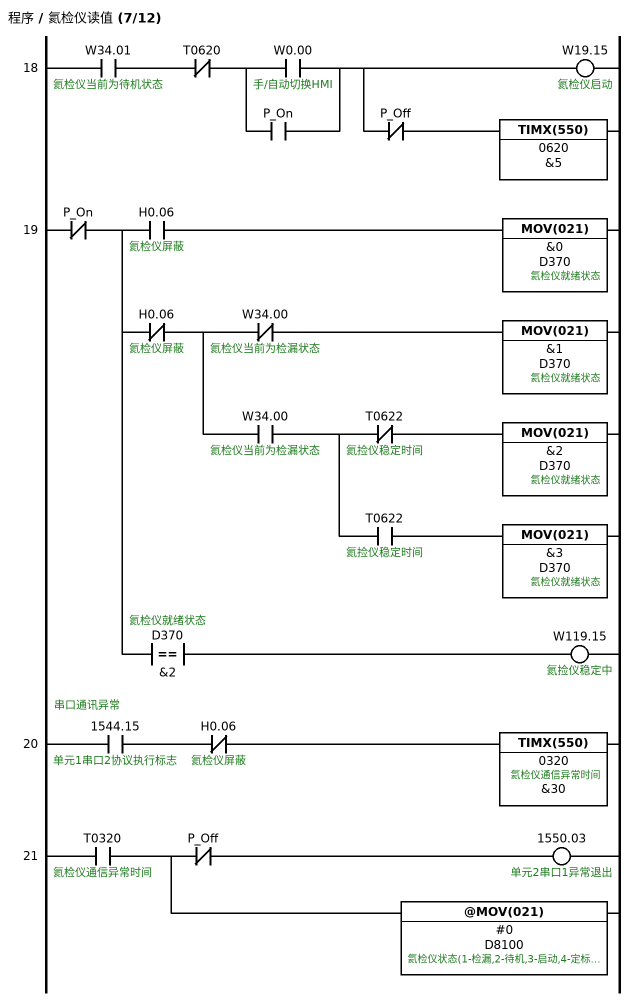
; [picture p168: 程序 / 氦检仪读值, rungs 18-21]
; rung 18
LD W34.01  ; 氦检仪当前为待机状态
ANDNOT T0620
LD W0.00  ; 手/自动切换HMI
OR P_On
ANDLD
OUT W19.15  ; 氦检仪启动
ANDNOT P_Off
TIMX(550) 0620 &5
; rung 19
LDNOT P_On
OUT TR0
AND H0.06  ; 氦检仪屏蔽
MOV(021) &0 D370  ; 氦检仪就绪状态
LD TR0
ANDNOT H0.06  ; 氦检仪屏蔽
OUT TR1
ANDNOT W34.00  ; 氦检仪当前为检漏状态
MOV(021) &1 D370  ; 氦检仪就绪状态
LD TR1
AND W34.00  ; 氦检仪当前为检漏状态
OUT TR1
ANDNOT T0622  ; 氦捡仪稳定时间
MOV(021) &2 D370  ; 氦检仪就绪状态
LD TR1
AND T0622  ; 氦捡仪稳定时间
MOV(021) &3 D370  ; 氦检仪就绪状态
LD TR0
AND=(300) D370 &2  ; 氦检仪就绪状态
OUT W119.15  ; 氦捡仪稳定中
; rung 20: 串口通讯异常
LD 1544.15  ; 单元1串口2协议执行标志
ANDNOT H0.06  ; 氦检仪屏蔽
TIMX(550) 0320 &30  ; 氦检仪通信异常时间
; rung 21
LD T0320  ; 氦检仪通信异常时间
OUT TR0
ANDNOT P_Off
OUT 1550.03  ; 单元2串口1异常退出
LD TR0
@MOV(021) #0 D8100  ; 氦检仪状态(1-检漏,2-待机,3-启动,4-定标,5-错误,6-暂停)

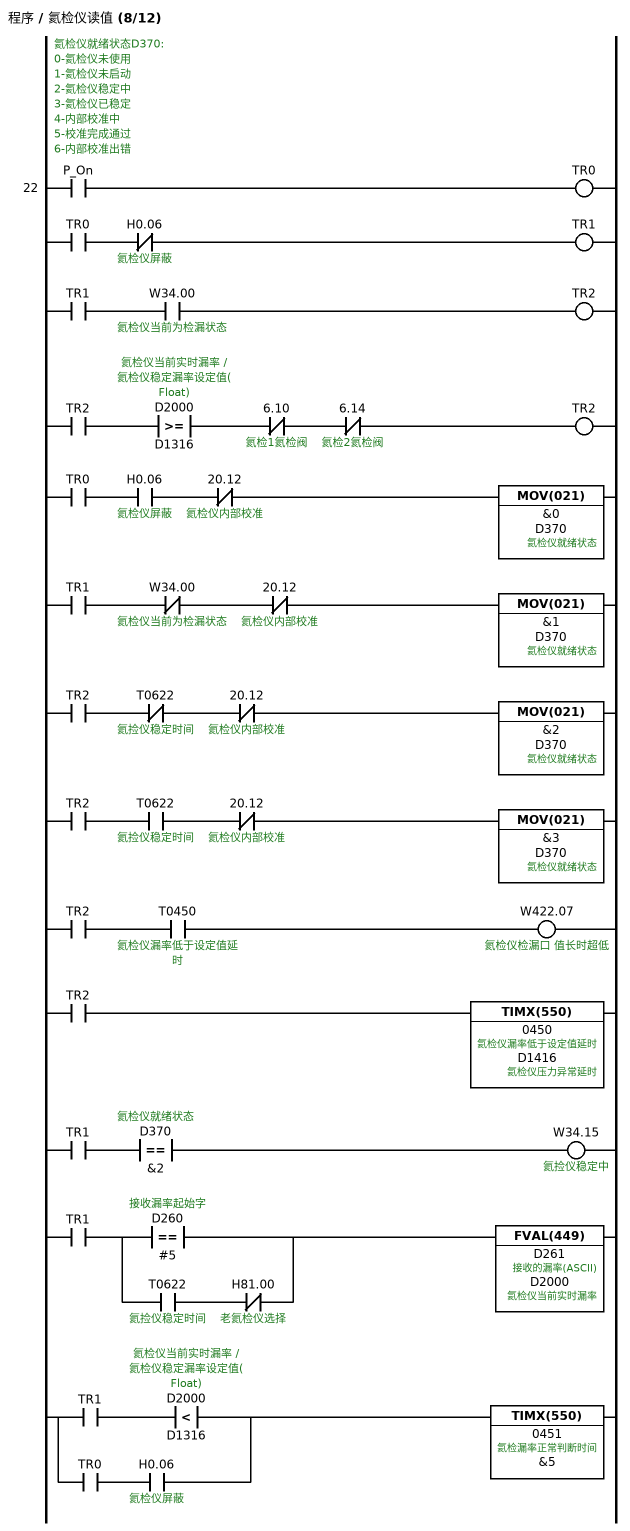
; rung 22: 氦检仪就绪状态D370: / 0-氦检仪未使用 / 1-氦检仪未启动 / 2-氦检仪稳定中 / 3-氦检仪已稳定 / 4-内部校准中 / 5-校准完成通过 / 6-内部校准出错
LD P_On
OUT TR0
AND H0.06  ; 氦检仪屏蔽
ANDNOT 20.12  ; 氦检仪内部校准
MOV(021) &0 D370  ; 氦检仪就绪状态
LD TR0
ANDNOT H0.06  ; 氦检仪屏蔽
OUT TR1
ANDNOT W34.00  ; 氦检仪当前为检漏状态
ANDNOT 20.12  ; 氦检仪内部校准
MOV(021) &1 D370  ; 氦检仪就绪状态
LD TR1
AND W34.00  ; 氦检仪当前为检漏状态
OUT TR2
ANDNOT T0622  ; 氦捡仪稳定时间
ANDNOT 20.12  ; 氦检仪内部校准
MOV(021) &2 D370  ; 氦检仪就绪状态
LD TR2
AND T0622  ; 氦捡仪稳定时间
ANDNOT 20.12  ; 氦检仪内部校准
MOV(021) &3 D370  ; 氦检仪就绪状态
LD TR2
AND>=F(334) D2000 D1316  ; 氦检仪当前实时漏率, 氦检仪稳定漏率设定值(Float)
ANDNOT 6.10  ; 氦检1氦检阀
ANDNOT 6.14  ; 氦检2氦检阀
OUT TR2
AND T0450  ; 氦检仪漏率低于设定值延时
OUT W422.07  ; 氦检仪检漏口 值长时超低
LD TR2
TIMX(550) 0450 D1416  ; 氦检仪压力异常延时, 氦检仪漏率低于设定值延时
LD TR1
AND=(300) D370 &2  ; 氦检仪就绪状态
OUT W34.15  ; 氦捡仪稳定中
LD TR1
LD=(300) D260 #5  ; 接收漏率起始字
LD T0622  ; 氦捡仪稳定时间
ANDNOT H81.00  ; 老氦检仪选择
ORLD
ANDLD
FVAL(449) D261 D2000  ; 接收的漏率(ASCII), 氦检仪当前实时漏率
LD TR1
AND<F(331) D2000 D1316  ; 氦检仪当前实时漏率, 氦检仪稳定漏率设定值(Float)
LD TR0
AND H0.06  ; 氦检仪屏蔽
ORLD
TIMX(550) 0451 &5  ; 氦检漏率正常判断时间

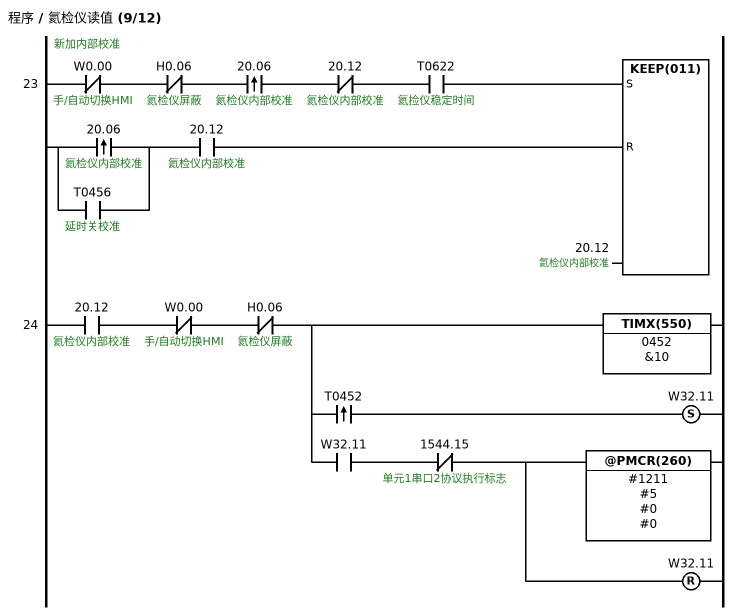
; rung 23: 新加内部校准
LDNOT W0.00  ; 手/自动切换HMI
ANDNOT H0.06  ; 氦检仪屏蔽
@AND 20.06  ; 氦检仪内部校准
ANDNOT 20.12  ; 氦检仪内部校准
AND T0622  ; 氦捡仪稳定时间
@LD 20.06  ; 氦检仪内部校准
OR T0456  ; 延时关校准
AND 20.12  ; 氦检仪内部校准
KEEP(011) 20.12  ; 氦检仪内部校准
; rung 24
LD 20.12  ; 氦检仪内部校准
ANDNOT W0.00  ; 手/自动切换HMI
ANDNOT H0.06  ; 氦检仪屏蔽
OUT TR0
TIMX(550) 0452 &10
@AND T0452
SET W32.11
LD TR0
AND W32.11
ANDNOT 1544.15  ; 单元1串口2协议执行标志
@PMCR(260) #1211 #5 #0 #0
RSET W32.11

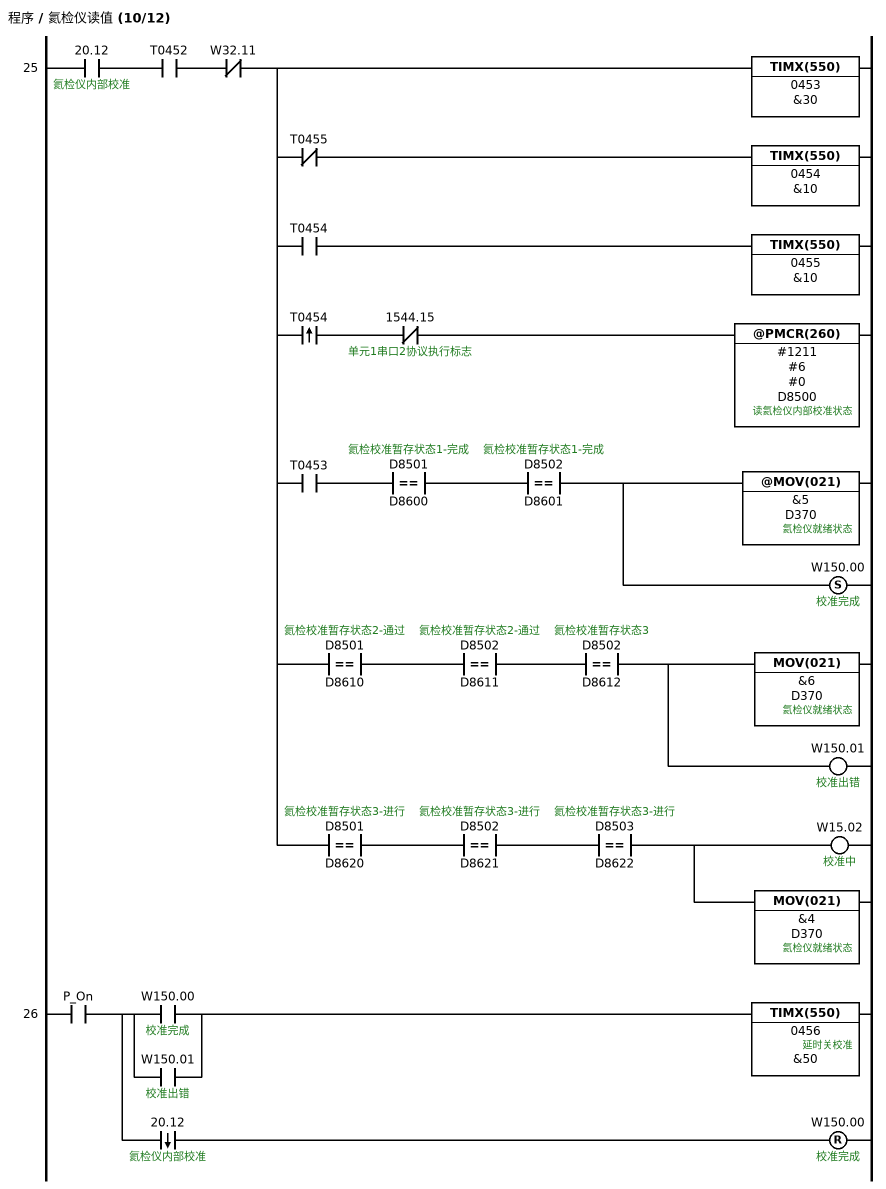
; rung 25
LD 20.12  ; 氦检仪内部校准
AND T0452
ANDNOT W32.11
OUT TR0
TIMX(550) 0453 &30
ANDNOT T0455
TIMX(550) 0454 &10
LD TR0
AND T0454
TIMX(550) 0455 &10
LD TR0
@AND T0454
ANDNOT 1544.15  ; 单元1串口2协议执行标志
@PMCR(260) #1211 #6 #0 D8500  ; 读氦检仪内部校准状态
LD TR0
AND T0453
AND=(300) D8501 D8600  ; 氦检校准暂存状态1-完成
AND=(300) D8502 D8601  ; 氦检校准暂存状态1-完成
@MOV(021) &5 D370  ; 氦检仪就绪状态
SET W150.00  ; 校准完成
LD TR0
AND=(300) D8501 D8610  ; 氦检校准暂存状态2-通过
AND=(300) D8502 D8611  ; 氦检校准暂存状态2-通过
AND=(300) D8502 D8612  ; 氦检校准暂存状态3
MOV(021) &6 D370  ; 氦检仪就绪状态
OUT W150.01  ; 校准出错
LD TR0
AND=(300) D8501 D8620  ; 氦检校准暂存状态3-进行
AND=(300) D8502 D8621  ; 氦检校准暂存状态3-进行
AND=(300) D8503 D8622  ; 氦检校准暂存状态3-进行
OUT W15.02  ; 校准中
MOV(021) &4 D370  ; 氦检仪就绪状态
; rung 26
LD P_On
OUT TR0
LD W150.00  ; 校准完成
OR W150.01  ; 校准出错
ANDLD
TIMX(550) 0456 &50  ; 延时关校准
LD TR0
%AND 20.12  ; 氦检仪内部校准
RSET W150.00  ; 校准完成

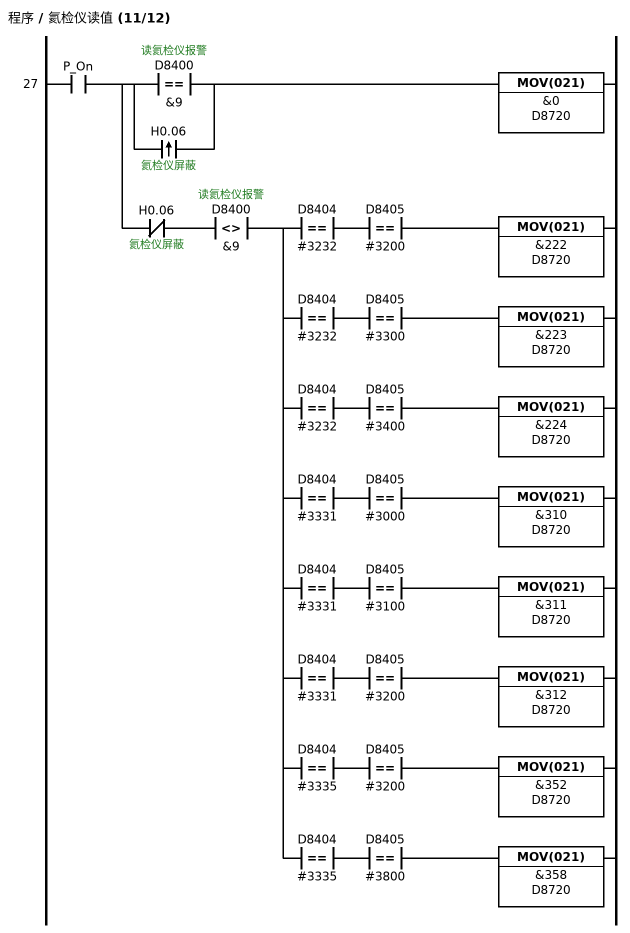
; rung 27
LD P_On
OUT TR0
LD=(300) D8400 &9  ; 读氦检仪报警
@OR H0.06  ; 氦检仪屏蔽
ANDLD
MOV(021) &0 D8720
LD TR0
ANDNOT H0.06  ; 氦检仪屏蔽
AND<>(305) D8400 &9  ; 读氦检仪报警
OUT TR0
AND=(300) D8404 #3232
AND=(300) D8405 #3200
MOV(021) &222 D8720
LD TR0
AND=(300) D8404 #3232
AND=(300) D8405 #3300
MOV(021) &223 D8720
LD TR0
AND=(300) D8404 #3232
AND=(300) D8405 #3400
MOV(021) &224 D8720
LD TR0
AND=(300) D8404 #3331
AND=(300) D8405 #3000
MOV(021) &310 D8720
LD TR0
AND=(300) D8404 #3331
AND=(300) D8405 #3100
MOV(021) &311 D8720
LD TR0
AND=(300) D8404 #3331
AND=(300) D8405 #3200
MOV(021) &312 D8720
LD TR0
AND=(300) D8404 #3335
AND=(300) D8405 #3200
MOV(021) &352 D8720
LD TR0
AND=(300) D8404 #3335
AND=(300) D8405 #3800
MOV(021) &358 D8720

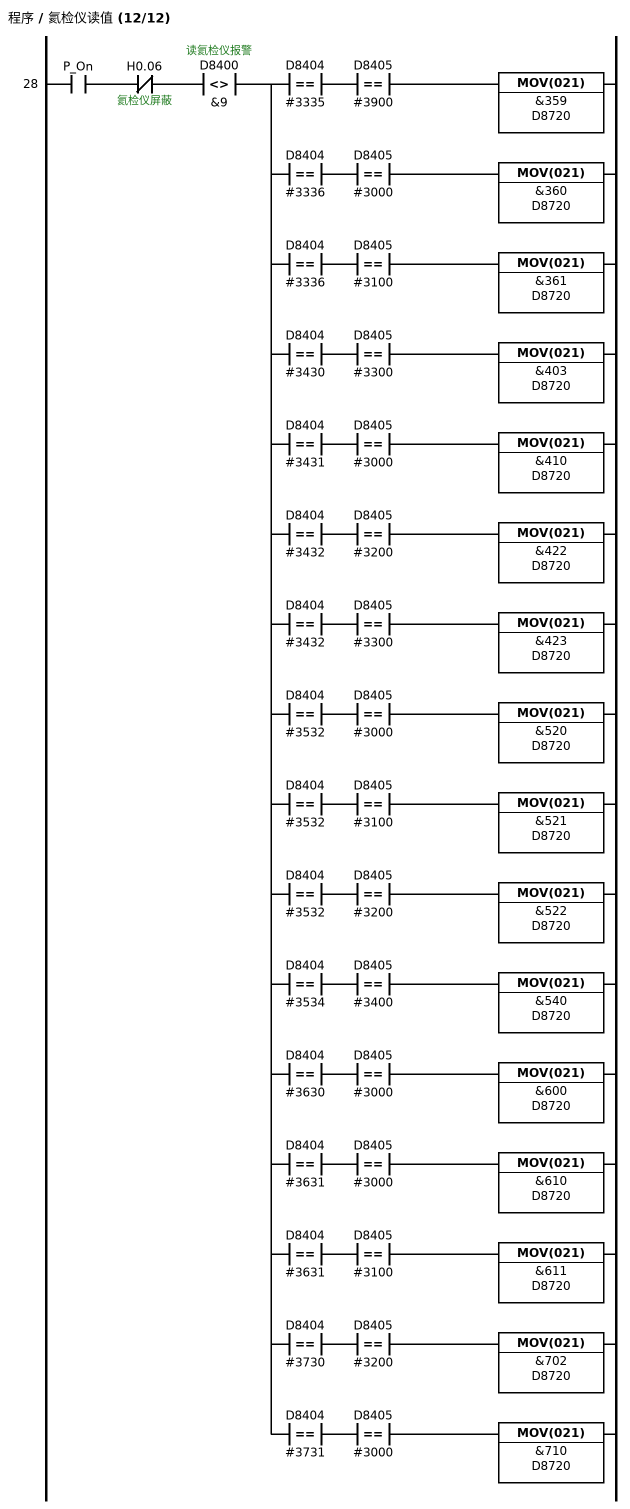
; rung 28
LD P_On
ANDNOT H0.06  ; 氦检仪屏蔽
AND<>(305) D8400 &9  ; 读氦检仪报警
OUT TR0
AND=(300) D8404 #3335
AND=(300) D8405 #3900
MOV(021) &359 D8720
LD TR0
AND=(300) D8404 #3336
AND=(300) D8405 #3000
MOV(021) &360 D8720
LD TR0
AND=(300) D8404 #3336
AND=(300) D8405 #3100
MOV(021) &361 D8720
LD TR0
AND=(300) D8404 #3430
AND=(300) D8405 #3300
MOV(021) &403 D8720
LD TR0
AND=(300) D8404 #3431
AND=(300) D8405 #3000
MOV(021) &410 D8720
LD TR0
AND=(300) D8404 #3432
AND=(300) D8405 #3200
MOV(021) &422 D8720
LD TR0
AND=(300) D8404 #3432
AND=(300) D8405 #3300
MOV(021) &423 D8720
LD TR0
AND=(300) D8404 #3532
AND=(300) D8405 #3000
MOV(021) &520 D8720
LD TR0
AND=(300) D8404 #3532
AND=(300) D8405 #3100
MOV(021) &521 D8720
LD TR0
AND=(300) D8404 #3532
AND=(300) D8405 #3200
MOV(021) &522 D8720
LD TR0
AND=(300) D8404 #3534
AND=(300) D8405 #3400
MOV(021) &540 D8720
LD TR0
AND=(300) D8404 #3630
AND=(300) D8405 #3000
MOV(021) &600 D8720
LD TR0
AND=(300) D8404 #3631
AND=(300) D8405 #3000
MOV(021) &610 D8720
LD TR0
AND=(300) D8404 #3631
AND=(300) D8405 #3100
MOV(021) &611 D8720
LD TR0
AND=(300) D8404 #3730
AND=(300) D8405 #3200
MOV(021) &702 D8720
LD TR0
AND=(300) D8404 #3731
AND=(300) D8405 #3000
MOV(021) &710 D8720

### Section 真空值及漏率标准转换

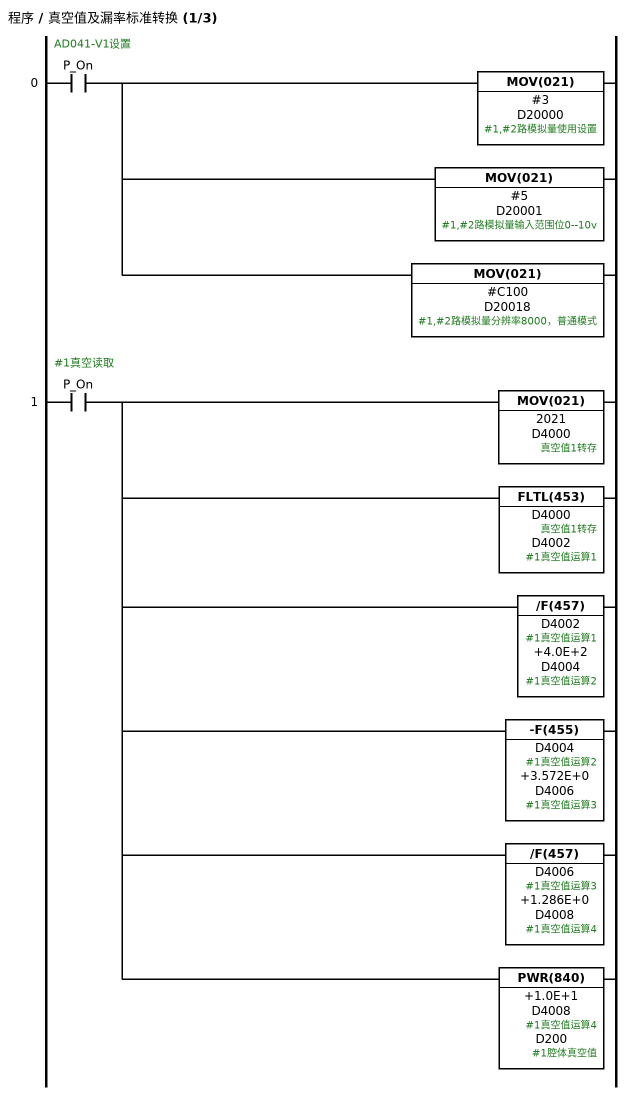
; rung 0: AD041-V1设置
LD P_On
MOV(021) #3 D20000  ; #1,#2路模拟量使用设置
MOV(021) #5 D20001  ; #1,#2路模拟量输入范围位0--10v
MOV(021) #C100 D20018  ; #1,#2路模拟量分辨率8000，普通模式
; rung 1: #1真空读取
LD P_On
MOV(021) 2021 D4000  ; 真空值1转存
FLTL(453) D4000 D4002  ; 真空值1转存, #1真空值运算1
/F(457) D4002 +4.0E+2 D4004  ; #1真空值运算1, #1真空值运算2
-F(455) D4004 +3.572E+0 D4006  ; #1真空值运算2, #1真空值运算3
/F(457) D4006 +1.286E+0 D4008  ; #1真空值运算3, #1真空值运算4
PWR(840) +1.0E+1 D4008 D200  ; #1真空值运算4, #1腔体真空值

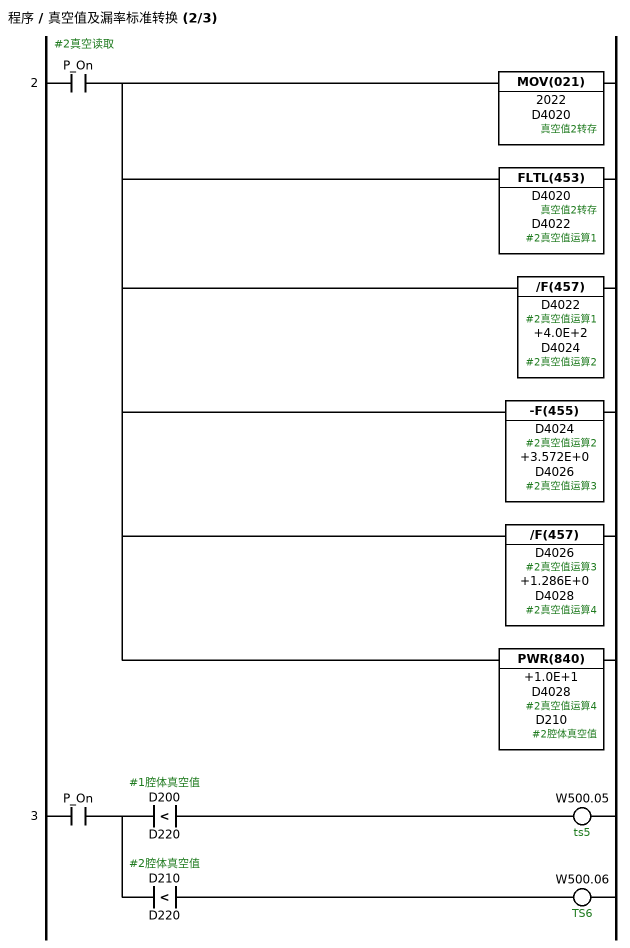
; rung 2: #2真空读取
LD P_On
MOV(021) 2022 D4020  ; 真空值2转存
FLTL(453) D4020 D4022  ; 真空值2转存, #2真空值运算1
/F(457) D4022 +4.0E+2 D4024  ; #2真空值运算1, #2真空值运算2
-F(455) D4024 +3.572E+0 D4026  ; #2真空值运算2, #2真空值运算3
/F(457) D4026 +1.286E+0 D4028  ; #2真空值运算3, #2真空值运算4
PWR(840) +1.0E+1 D4028 D210  ; #2真空值运算4, #2腔体真空值
; rung 3
LD P_On
OUT TR0
AND<F(331) D200 D220  ; #1腔体真空值
OUT W500.05  ; ts5
LD TR0
AND<F(331) D210 D220  ; #2腔体真空值
OUT W500.06  ; TS6

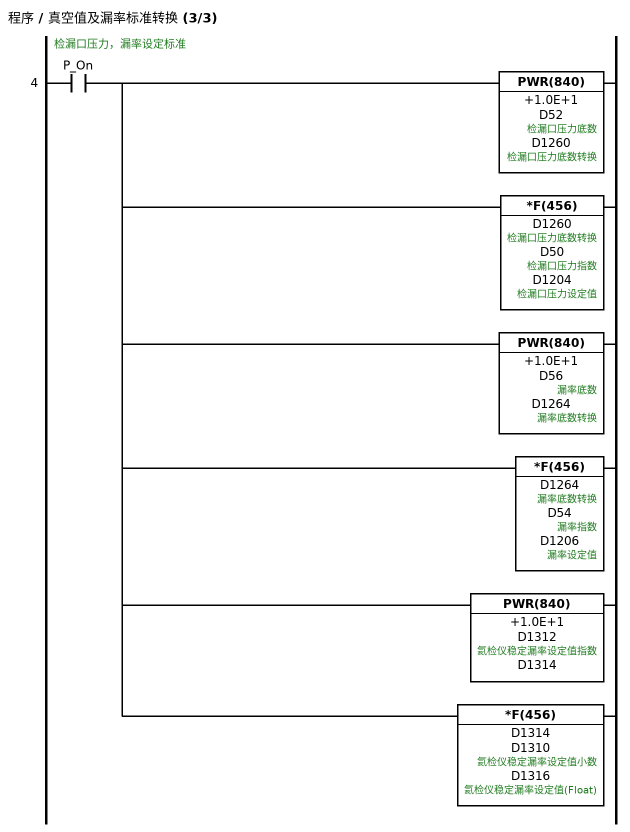
; rung 4: 检漏口压力，漏率设定标准
LD P_On
PWR(840) +1.0E+1 D52 D1260  ; 检漏口压力底数, 检漏口压力底数转换
*F(456) D1260 D50 D1204  ; 检漏口压力底数转换, 检漏口压力指数, 检漏口压力设定值
PWR(840) +1.0E+1 D56 D1264  ; 漏率底数, 漏率底数转换
*F(456) D1264 D54 D1206  ; 漏率底数转换, 漏率指数, 漏率设定值
PWR(840) +1.0E+1 D1312 D1314  ; 氦检仪稳定漏率设定值指数
*F(456) D1314 D1310 D1316  ; 氦检仪稳定漏率设定值小数, 氦检仪稳定漏率设定值(Float)

### Section 腔体自检

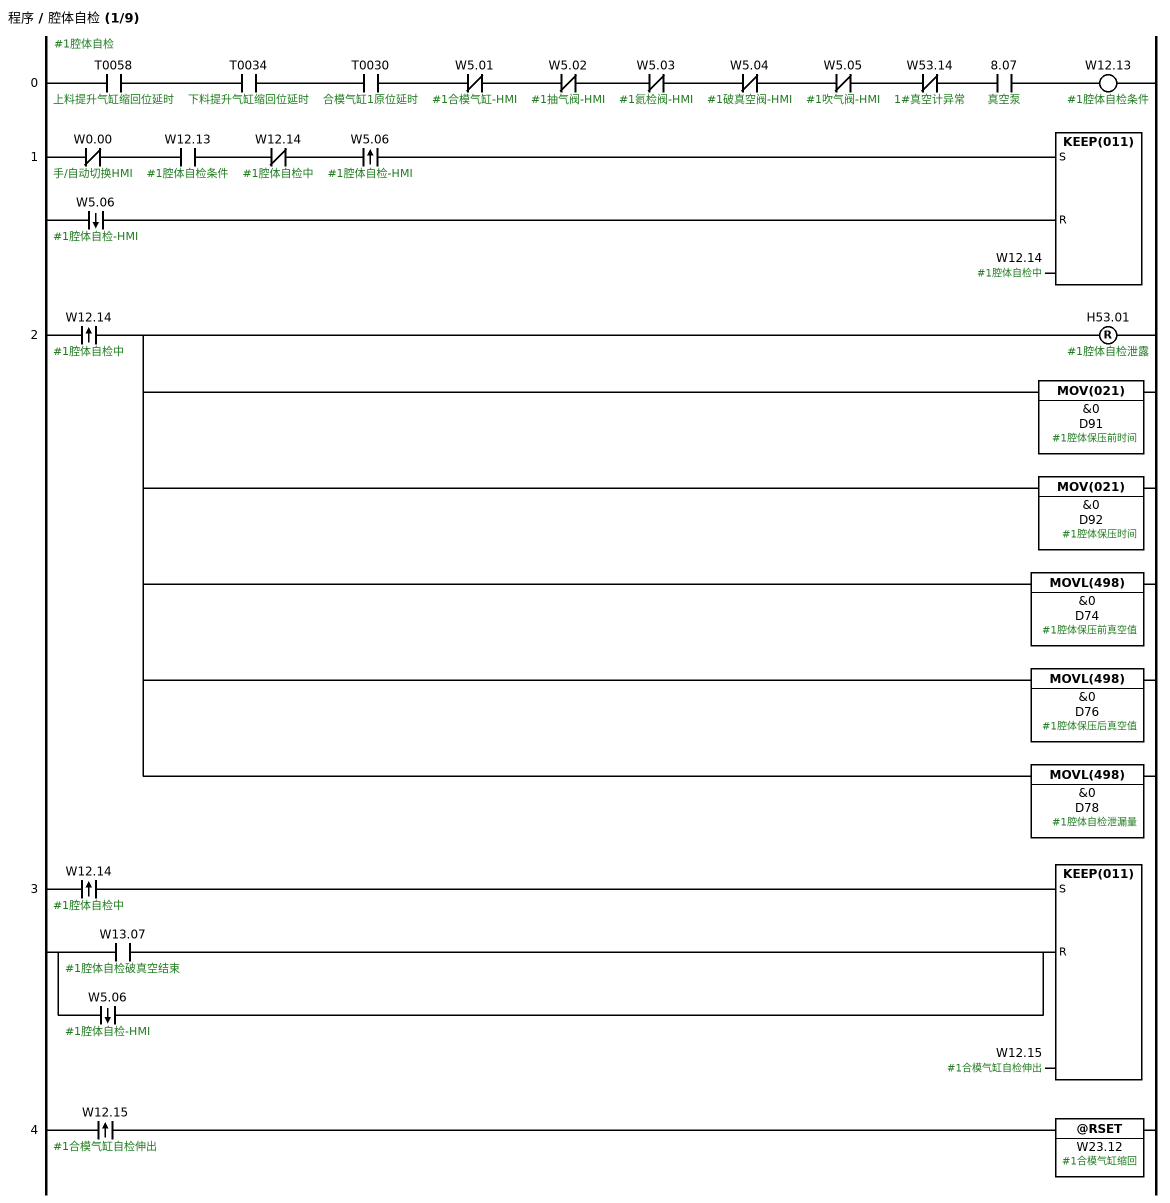
; rung 0: #1腔体自检
LD T0058  ; 上料提升气缸缩回位延时
AND T0034  ; 下料提升气缸缩回位延时
AND T0030  ; 合模气缸1原位延时
ANDNOT W5.01  ; #1合模气缸-HMI
ANDNOT W5.02  ; #1抽气阀-HMI
ANDNOT W5.03  ; #1氦检阀-HMI
ANDNOT W5.04  ; #1破真空阀-HMI
ANDNOT W5.05  ; #1吹气阀-HMI
ANDNOT W53.14  ; 1#真空计异常
AND 8.07  ; 真空泵
OUT W12.13  ; #1腔体自检条件
; rung 1
LDNOT W0.00  ; 手/自动切换HMI
AND W12.13  ; #1腔体自检条件
ANDNOT W12.14  ; #1腔体自检中
@AND W5.06  ; #1腔体自检-HMI
%LD W5.06  ; #1腔体自检-HMI
KEEP(011) W12.14  ; #1腔体自检中
; rung 2
@LD W12.14  ; #1腔体自检中
RSET H53.01  ; #1腔体自检泄露
MOV(021) &0 D91  ; #1腔体保压前时间
MOV(021) &0 D92  ; #1腔体保压时间
MOVL(498) &0 D74  ; #1腔体保压前真空值
MOVL(498) &0 D76  ; #1腔体保压后真空值
MOVL(498) &0 D78  ; #1腔体自检泄漏量
; rung 3
@LD W12.14  ; #1腔体自检中
LD W13.07  ; #1腔体自检破真空结束
%OR W5.06  ; #1腔体自检-HMI
KEEP(011) W12.15  ; #1合模气缸自检伸出
; rung 4
@LD W12.15  ; #1合模气缸自检伸出
@RSET W23.12  ; #1合模气缸缩回

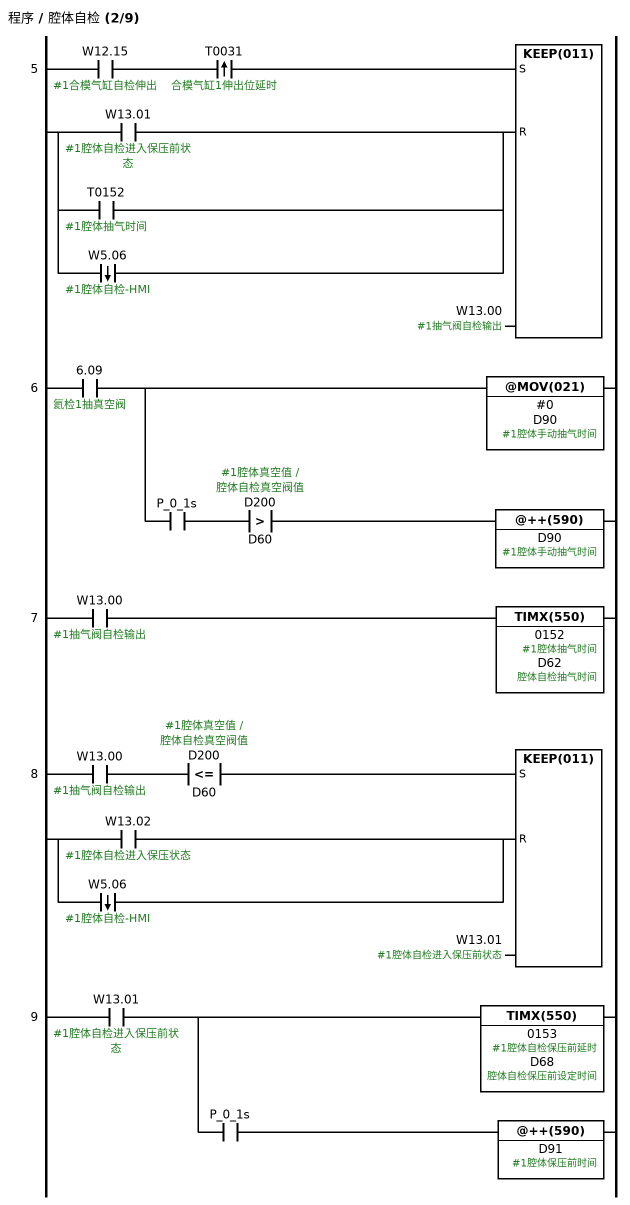
; rung 5
LD W12.15  ; #1合模气缸自检伸出
@AND T0031  ; 合模气缸1伸出位延时
LD W13.01  ; #1腔体自检进入保压前状态
OR T0152  ; #1腔体抽气时间
%OR W5.06  ; #1腔体自检-HMI
KEEP(011) W13.00  ; #1抽气阀自检输出
; rung 6
LD 6.09  ; 氦检1抽真空阀
@MOV(021) #0 D90  ; #1腔体手动抽气时间
AND P_0_1s
AND>F(333) D200 D60  ; #1腔体真空值, 腔体自检真空阀值
@++(590) D90  ; #1腔体手动抽气时间
; rung 7
LD W13.00  ; #1抽气阀自检输出
TIMX(550) 0152 D62  ; 腔体自检抽气时间, #1腔体抽气时间
; rung 8
LD W13.00  ; #1抽气阀自检输出
AND<=F(332) D200 D60  ; #1腔体真空值, 腔体自检真空阀值
LD W13.02  ; #1腔体自检进入保压状态
%OR W5.06  ; #1腔体自检-HMI
KEEP(011) W13.01  ; #1腔体自检进入保压前状态
; rung 9
LD W13.01  ; #1腔体自检进入保压前状态
TIMX(550) 0153 D68  ; 腔体自检保压前设定时间, #1腔体自检保压前延时
AND P_0_1s
@++(590) D91  ; #1腔体保压前时间

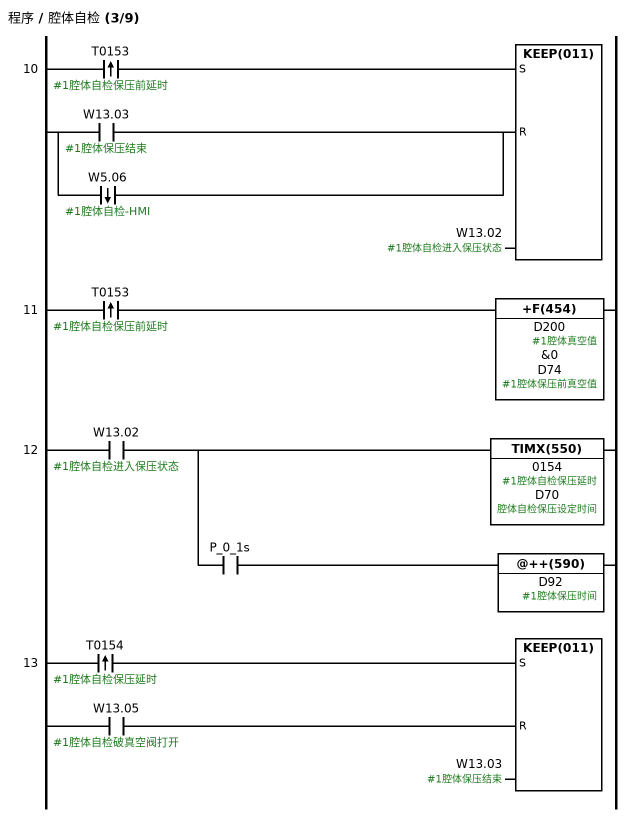
; rung 10
@LD T0153  ; #1腔体自检保压前延时
LD W13.03  ; #1腔体保压结束
%OR W5.06  ; #1腔体自检-HMI
KEEP(011) W13.02  ; #1腔体自检进入保压状态
; rung 11
@LD T0153  ; #1腔体自检保压前延时
+F(454) D200 &0 D74  ; #1腔体真空值, #1腔体保压前真空值
; rung 12
LD W13.02  ; #1腔体自检进入保压状态
TIMX(550) 0154 D70  ; 腔体自检保压设定时间, #1腔体自检保压延时
AND P_0_1s
@++(590) D92  ; #1腔体保压时间
; rung 13
@LD T0154  ; #1腔体自检保压延时
LD W13.05  ; #1腔体自检破真空阀打开
KEEP(011) W13.03  ; #1腔体保压结束

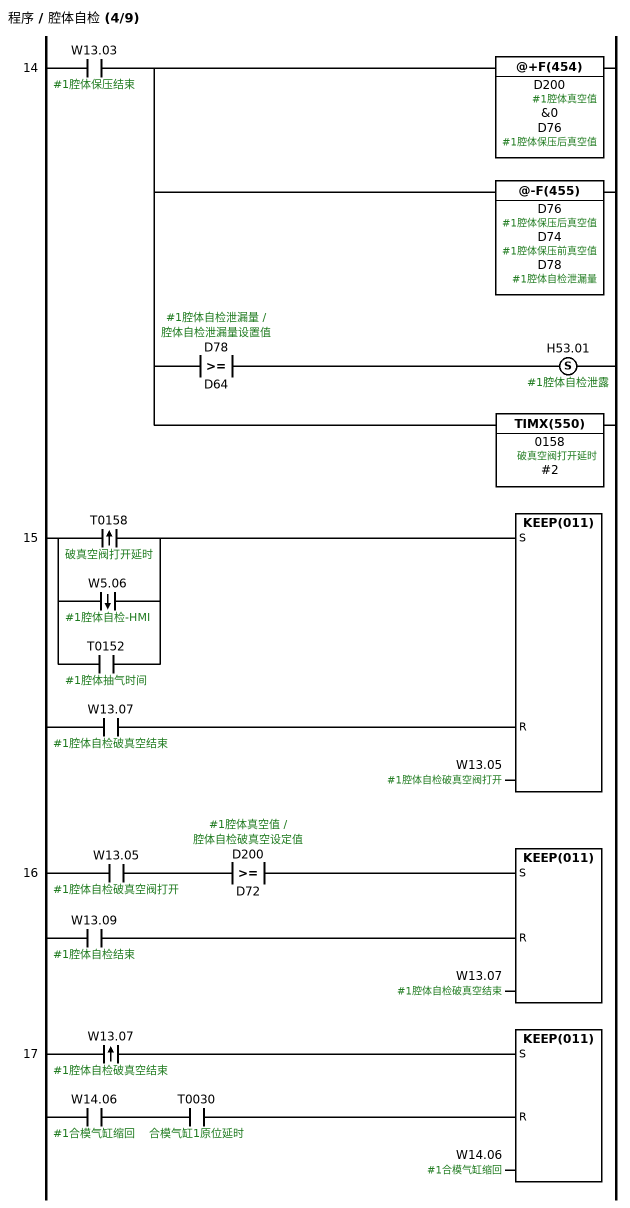
; rung 14
LD W13.03  ; #1腔体保压结束
OUT TR0
@+F(454) D200 &0 D76  ; #1腔体真空值, #1腔体保压后真空值
@-F(455) D76 D74 D78  ; #1腔体保压后真空值, #1腔体保压前真空值, #1腔体自检泄漏量
AND>=F(334) D78 D64  ; #1腔体自检泄漏量, 腔体自检泄漏量设置值
SET H53.01  ; #1腔体自检泄露
LD TR0
TIMX(550) 0158 #2  ; 破真空阀打开延时
; rung 15
@LD T0158  ; 破真空阀打开延时
%OR W5.06  ; #1腔体自检-HMI
OR T0152  ; #1腔体抽气时间
LD W13.07  ; #1腔体自检破真空结束
KEEP(011) W13.05  ; #1腔体自检破真空阀打开
; rung 16
LD W13.05  ; #1腔体自检破真空阀打开
AND>=F(334) D200 D72  ; #1腔体真空值, 腔体自检破真空设定值
LD W13.09  ; #1腔体自检结束
KEEP(011) W13.07  ; #1腔体自检破真空结束
; rung 17
@LD W13.07  ; #1腔体自检破真空结束
LD W14.06  ; #1合模气缸缩回
AND T0030  ; 合模气缸1原位延时
KEEP(011) W14.06  ; #1合模气缸缩回

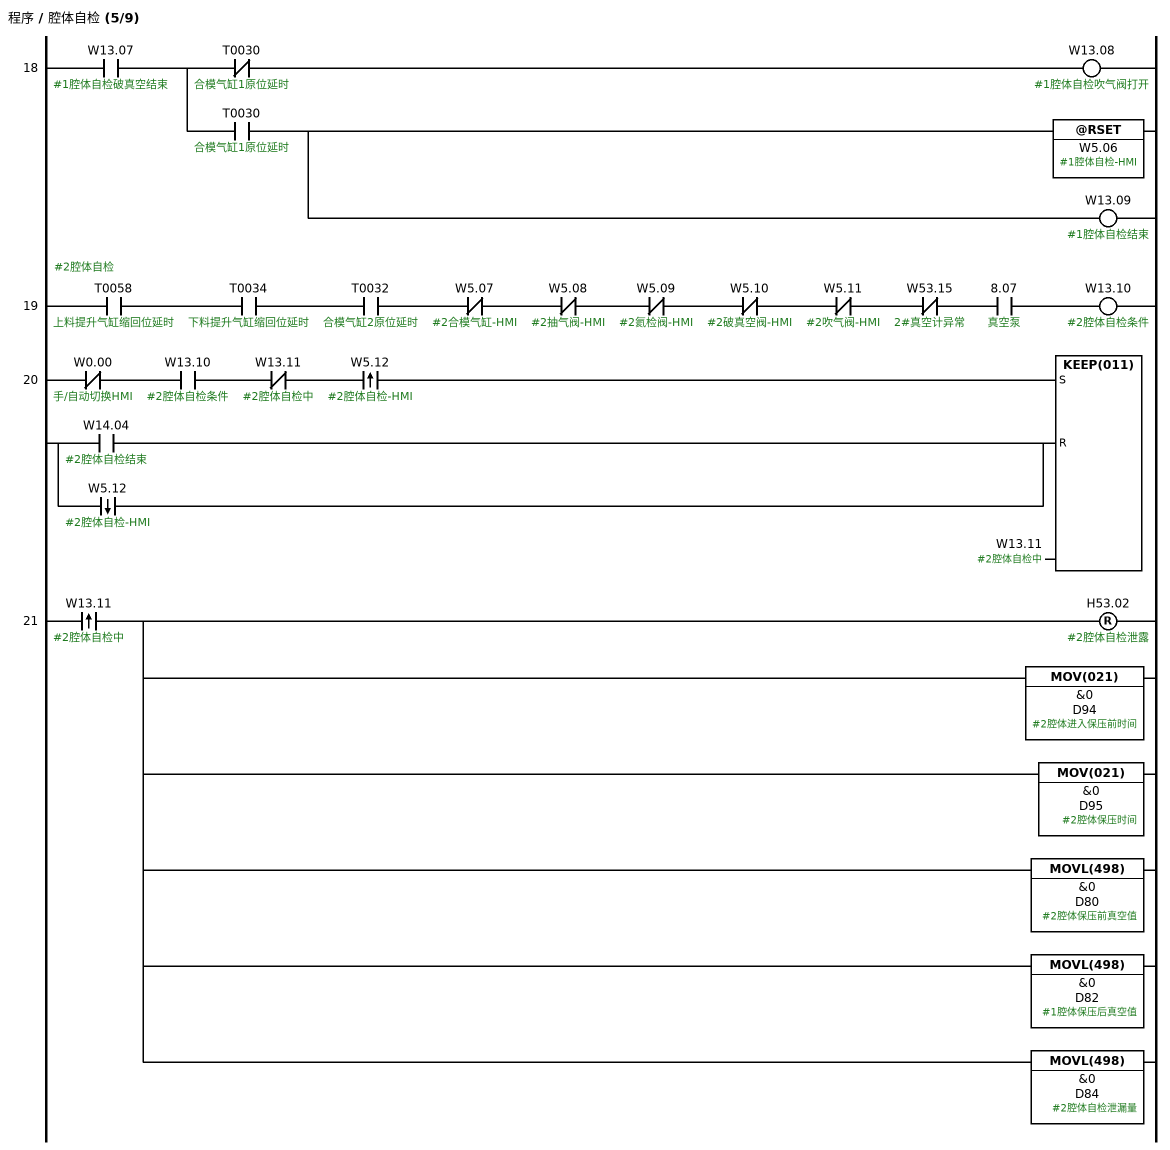
; rung 18
LD W13.07  ; #1腔体自检破真空结束
OUT TR0
ANDNOT T0030  ; 合模气缸1原位延时
OUT W13.08  ; #1腔体自检吹气阀打开
LD TR0
AND T0030  ; 合模气缸1原位延时
@RSET W5.06  ; #1腔体自检-HMI
OUT W13.09  ; #1腔体自检结束
; rung 19: #2腔体自检
LD T0058  ; 上料提升气缸缩回位延时
AND T0034  ; 下料提升气缸缩回位延时
AND T0032  ; 合模气缸2原位延时
ANDNOT W5.07  ; #2合模气缸-HMI
ANDNOT W5.08  ; #2抽气阀-HMI
ANDNOT W5.09  ; #2氦检阀-HMI
ANDNOT W5.10  ; #2破真空阀-HMI
ANDNOT W5.11  ; #2吹气阀-HMI
ANDNOT W53.15  ; 2#真空计异常
AND 8.07  ; 真空泵
OUT W13.10  ; #2腔体自检条件
; rung 20
LDNOT W0.00  ; 手/自动切换HMI
AND W13.10  ; #2腔体自检条件
ANDNOT W13.11  ; #2腔体自检中
@AND W5.12  ; #2腔体自检-HMI
LD W14.04  ; #2腔体自检结束
%OR W5.12  ; #2腔体自检-HMI
KEEP(011) W13.11  ; #2腔体自检中
; rung 21
@LD W13.11  ; #2腔体自检中
RSET H53.02  ; #2腔体自检泄露
MOV(021) &0 D94  ; #2腔体进入保压前时间
MOV(021) &0 D95  ; #2腔体保压时间
MOVL(498) &0 D80  ; #2腔体保压前真空值
MOVL(498) &0 D82  ; #1腔体保压后真空值
MOVL(498) &0 D84  ; #2腔体自检泄漏量

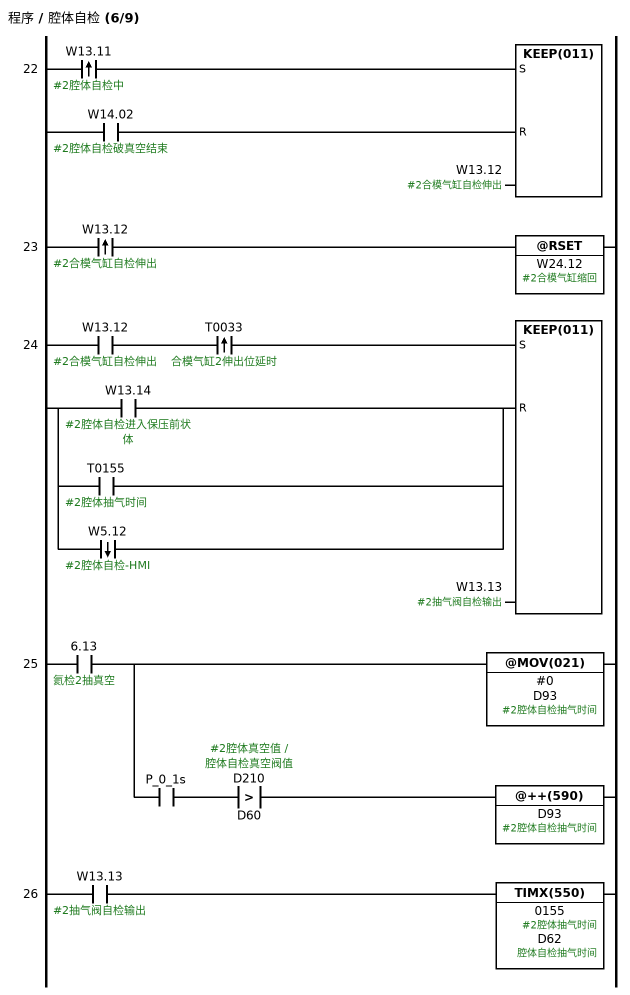
; rung 22
@LD W13.11  ; #2腔体自检中
LD W14.02  ; #2腔体自检破真空结束
KEEP(011) W13.12  ; #2合模气缸自检伸出
; rung 23
@LD W13.12  ; #2合模气缸自检伸出
@RSET W24.12  ; #2合模气缸缩回
; rung 24
LD W13.12  ; #2合模气缸自检伸出
@AND T0033  ; 合模气缸2伸出位延时
LD W13.14  ; #2腔体自检进入保压前状体
OR T0155  ; #2腔体抽气时间
%OR W5.12  ; #2腔体自检-HMI
KEEP(011) W13.13  ; #2抽气阀自检输出
; rung 25
LD 6.13  ; 氦检2抽真空
@MOV(021) #0 D93  ; #2腔体自检抽气时间
AND P_0_1s
AND>F(333) D210 D60  ; #2腔体真空值, 腔体自检真空阀值
@++(590) D93  ; #2腔体自检抽气时间
; rung 26
LD W13.13  ; #2抽气阀自检输出
TIMX(550) 0155 D62  ; 腔体自检抽气时间, #2腔体抽气时间

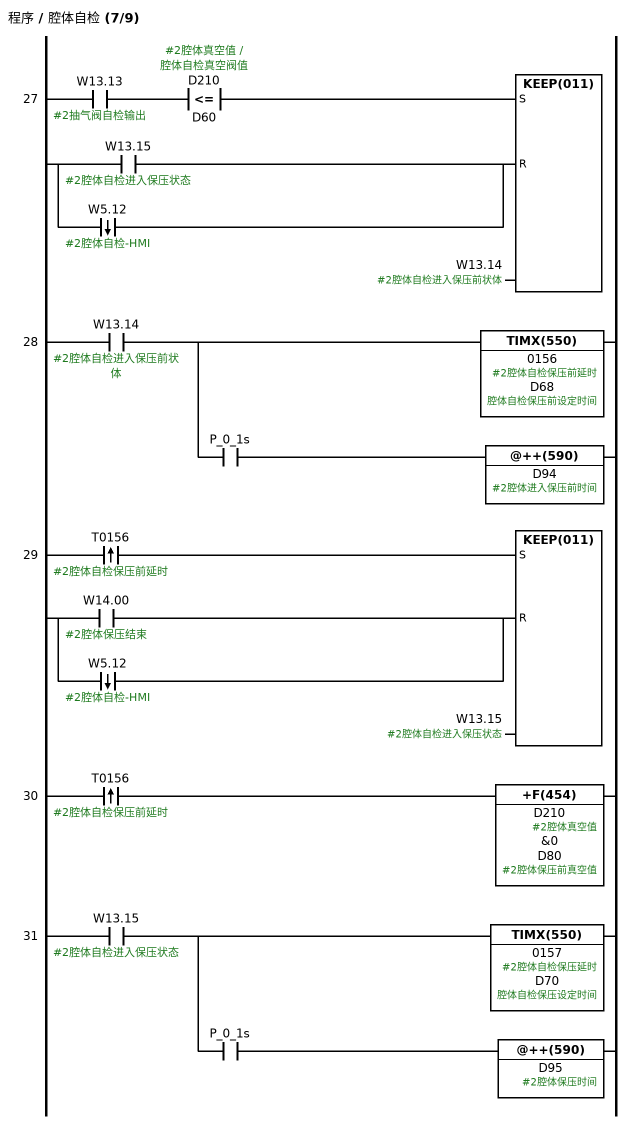
; rung 27
LD W13.13  ; #2抽气阀自检输出
AND<=F(332) D210 D60  ; #2腔体真空值, 腔体自检真空阀值
LD W13.15  ; #2腔体自检进入保压状态
%OR W5.12  ; #2腔体自检-HMI
KEEP(011) W13.14  ; #2腔体自检进入保压前状体
; rung 28
LD W13.14  ; #2腔体自检进入保压前状体
TIMX(550) 0156 D68  ; 腔体自检保压前设定时间, #2腔体自检保压前延时
AND P_0_1s
@++(590) D94  ; #2腔体进入保压前时间
; rung 29
@LD T0156  ; #2腔体自检保压前延时
LD W14.00  ; #2腔体保压结束
%OR W5.12  ; #2腔体自检-HMI
KEEP(011) W13.15  ; #2腔体自检进入保压状态
; rung 30
@LD T0156  ; #2腔体自检保压前延时
+F(454) D210 &0 D80  ; #2腔体真空值, #2腔体保压前真空值
; rung 31
LD W13.15  ; #2腔体自检进入保压状态
TIMX(550) 0157 D70  ; 腔体自检保压设定时间, #2腔体自检保压延时
AND P_0_1s
@++(590) D95  ; #2腔体保压时间

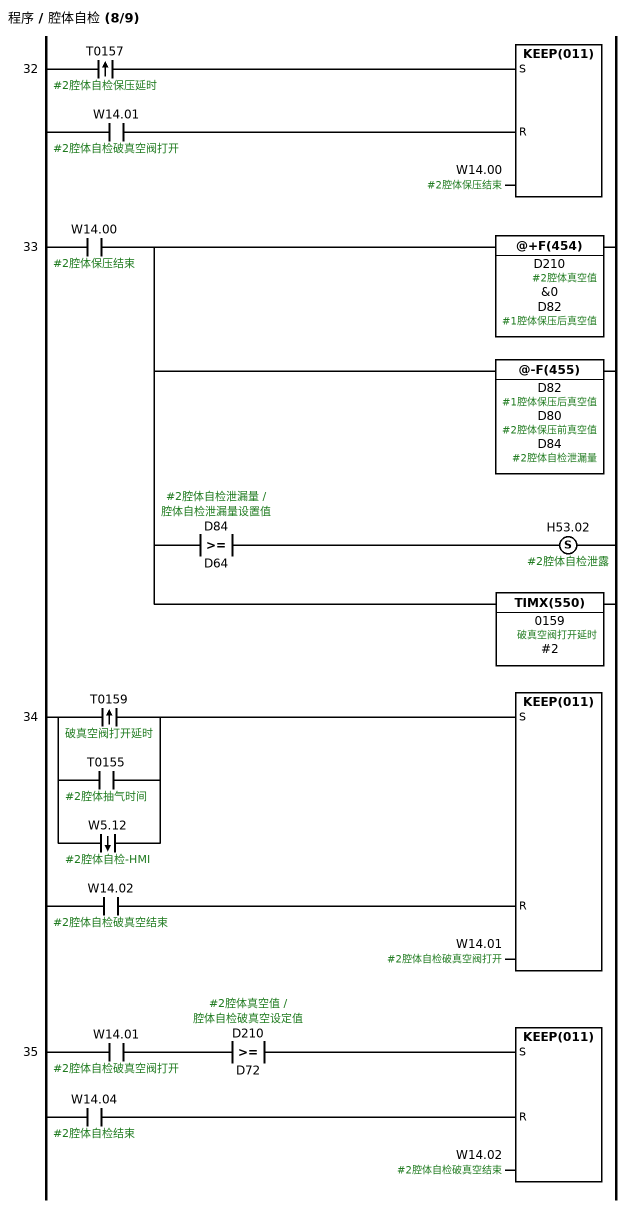
; rung 32
@LD T0157  ; #2腔体自检保压延时
LD W14.01  ; #2腔体自检破真空阀打开
KEEP(011) W14.00  ; #2腔体保压结束
; rung 33
LD W14.00  ; #2腔体保压结束
OUT TR0
@+F(454) D210 &0 D82  ; #2腔体真空值, #1腔体保压后真空值
@-F(455) D82 D80 D84  ; #1腔体保压后真空值, #2腔体保压前真空值, #2腔体自检泄漏量
AND>=F(334) D84 D64  ; #2腔体自检泄漏量, 腔体自检泄漏量设置值
SET H53.02  ; #2腔体自检泄露
LD TR0
TIMX(550) 0159 #2  ; 破真空阀打开延时
; rung 34
@LD T0159  ; 破真空阀打开延时
OR T0155  ; #2腔体抽气时间
%OR W5.12  ; #2腔体自检-HMI
LD W14.02  ; #2腔体自检破真空结束
KEEP(011) W14.01  ; #2腔体自检破真空阀打开
; rung 35
LD W14.01  ; #2腔体自检破真空阀打开
AND>=F(334) D210 D72  ; #2腔体真空值, 腔体自检破真空设定值
LD W14.04  ; #2腔体自检结束
KEEP(011) W14.02  ; #2腔体自检破真空结束

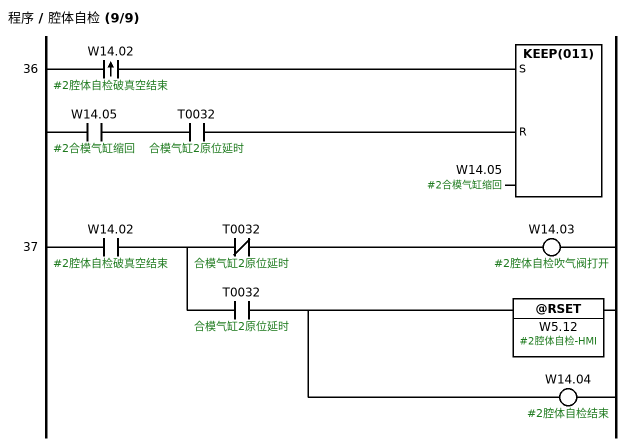
; rung 36
@LD W14.02  ; #2腔体自检破真空结束
LD W14.05  ; #2合模气缸缩回
AND T0032  ; 合模气缸2原位延时
KEEP(011) W14.05  ; #2合模气缸缩回
; rung 37
LD W14.02  ; #2腔体自检破真空结束
OUT TR0
ANDNOT T0032  ; 合模气缸2原位延时
OUT W14.03  ; #2腔体自检吹气阀打开
LD TR0
AND T0032  ; 合模气缸2原位延时
@RSET W5.12  ; #2腔体自检-HMI
OUT W14.04  ; #2腔体自检结束

### Section 报警

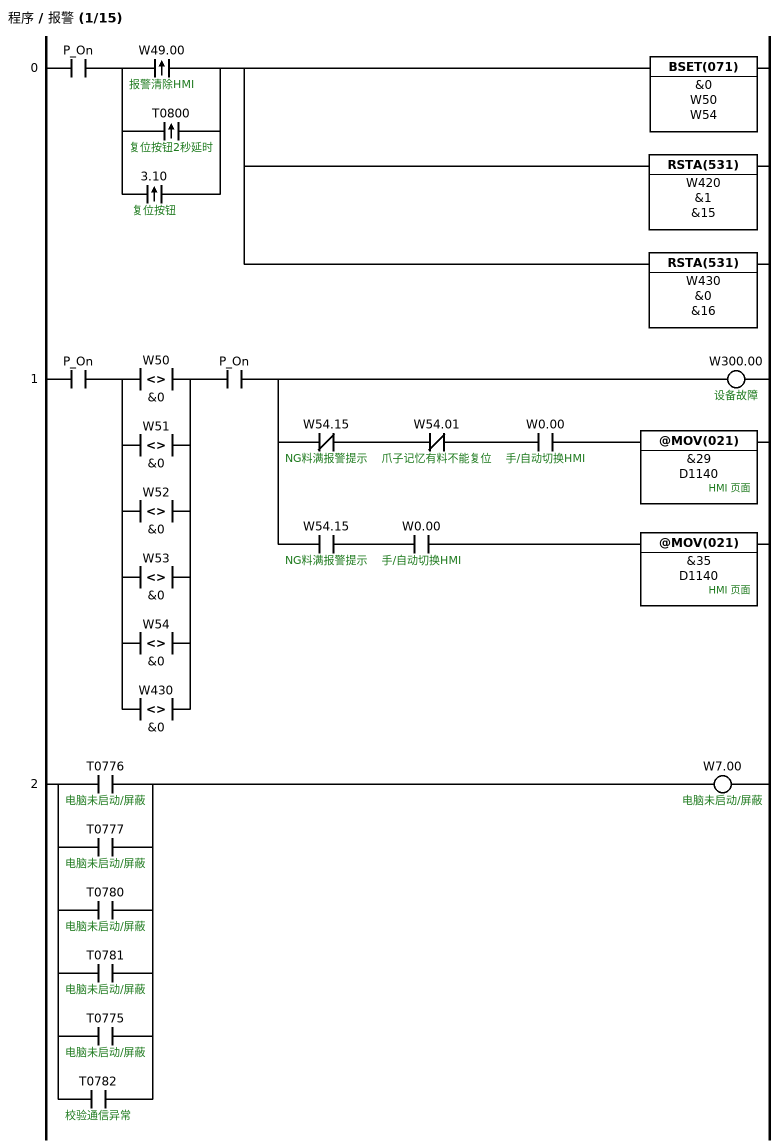
; rung 0
LD P_On
@LD W49.00  ; 报警清除HMI
@OR T0800  ; 复位按钮2秒延时
@OR 3.10  ; 复位按钮
ANDLD
BSET(071) &0 W50 W54
RSTA(531) W420 &1 &15
RSTA(531) W430 &0 &16
; rung 1
LD P_On
LD<>(305) W50 &0
OR<>(305) W51 &0
OR<>(305) W52 &0
OR<>(305) W53 &0
OR<>(305) W54 &0
OR<>(305) W430 &0
ANDLD
AND P_On
OUT TR0
OUT W300.00  ; 设备故障
ANDNOT W54.15  ; NG料满报警提示
ANDNOT W54.01  ; 爪子记忆有料不能复位
AND W0.00  ; 手/自动切换HMI
@MOV(021) &29 D1140  ; HMI 页面
LD TR0
AND W54.15  ; NG料满报警提示
AND W0.00  ; 手/自动切换HMI
@MOV(021) &35 D1140  ; HMI 页面
; rung 2
LD T0776  ; 电脑未启动/屏蔽
OR T0777  ; 电脑未启动/屏蔽
OR T0780  ; 电脑未启动/屏蔽
OR T0781  ; 电脑未启动/屏蔽
OR T0775  ; 电脑未启动/屏蔽
OR T0782  ; 校验通信异常
OUT W7.00  ; 电脑未启动/屏蔽

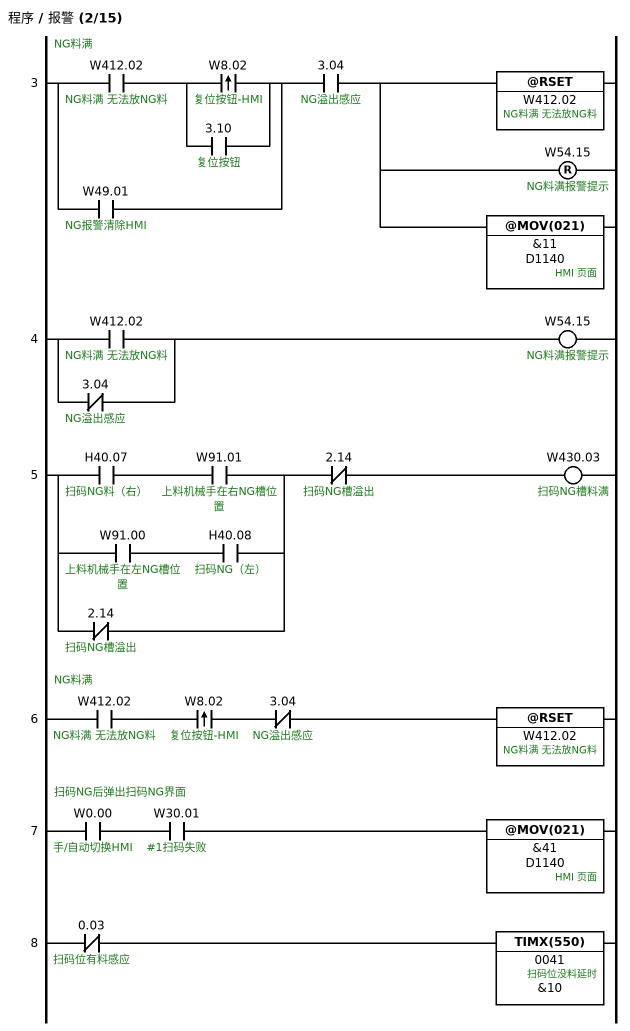
; rung 3: NG料满
LD W412.02  ; NG料满 无法放NG料
@LD W8.02  ; 复位按钮-HMI
OR 3.10  ; 复位按钮
ANDLD
OR W49.01  ; NG报警清除HMI
AND 3.04  ; NG溢出感应
@RSET W412.02  ; NG料满 无法放NG料
RSET W54.15  ; NG料满报警提示
@MOV(021) &11 D1140  ; HMI 页面
; rung 4
LD W412.02  ; NG料满 无法放NG料
ORNOT 3.04  ; NG溢出感应
OUT W54.15  ; NG料满报警提示
; rung 5
LD H40.07  ; 扫码NG料（右）
AND W91.01  ; 上料机械手在右NG槽位置
LD W91.00  ; 上料机械手在左NG槽位置
AND H40.08  ; 扫码NG（左）
ORLD
ORNOT 2.14  ; 扫码NG槽溢出
ANDNOT 2.14  ; 扫码NG槽溢出
OUT W430.03  ; 扫码NG槽料满
; rung 6: NG料满
LD W412.02  ; NG料满 无法放NG料
@AND W8.02  ; 复位按钮-HMI
ANDNOT 3.04  ; NG溢出感应
@RSET W412.02  ; NG料满 无法放NG料
; rung 7: 扫码NG后弹出扫码NG界面
LD W0.00  ; 手/自动切换HMI
AND W30.01  ; #1扫码失败
@MOV(021) &41 D1140  ; HMI 页面
; rung 8
LDNOT 0.03  ; 扫码位有料感应
TIMX(550) 0041 &10  ; 扫码位没料延时

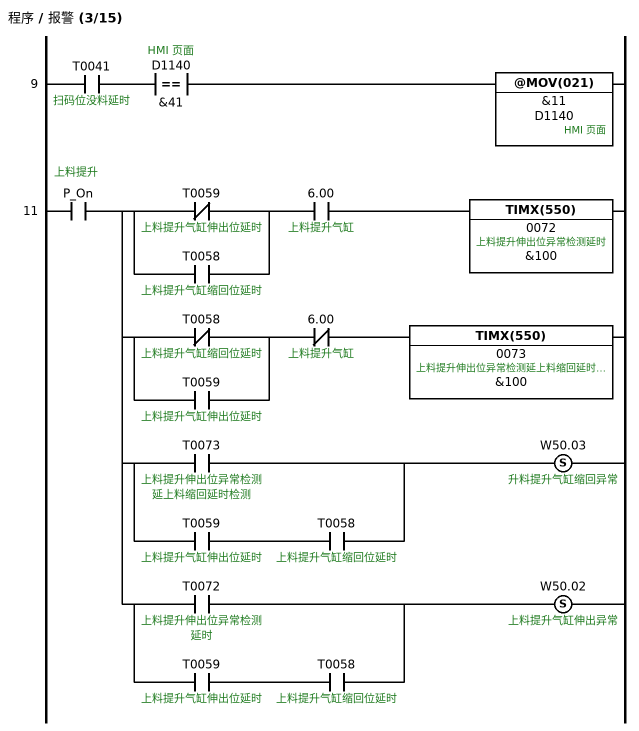
; rung 9
LD T0041  ; 扫码位没料延时
AND=(300) D1140 &41  ; HMI 页面
@MOV(021) &11 D1140  ; HMI 页面
; rung 11: 上料提升
LD P_On
OUT TR0
LDNOT T0059  ; 上料提升气缸伸出位延时
OR T0058  ; 上料提升气缸缩回位延时
ANDLD
AND 6.00  ; 上料提升气缸
TIMX(550) 0072 &100  ; 上料提升伸出位异常检测延时
LD TR0
LDNOT T0058  ; 上料提升气缸缩回位延时
OR T0059  ; 上料提升气缸伸出位延时
ANDLD
ANDNOT 6.00  ; 上料提升气缸
TIMX(550) 0073 &100  ; 上料提升伸出位异常检测延上料缩回延时检测
LD TR0
LD T0073  ; 上料提升伸出位异常检测延上料缩回延时检测
LD T0059  ; 上料提升气缸伸出位延时
AND T0058  ; 上料提升气缸缩回位延时
ORLD
ANDLD
SET W50.03  ; 升料提升气缸缩回异常
LD TR0
LD T0072  ; 上料提升伸出位异常检测延时
LD T0059  ; 上料提升气缸伸出位延时
AND T0058  ; 上料提升气缸缩回位延时
ORLD
ANDLD
SET W50.02  ; 上料提升气缸伸出异常

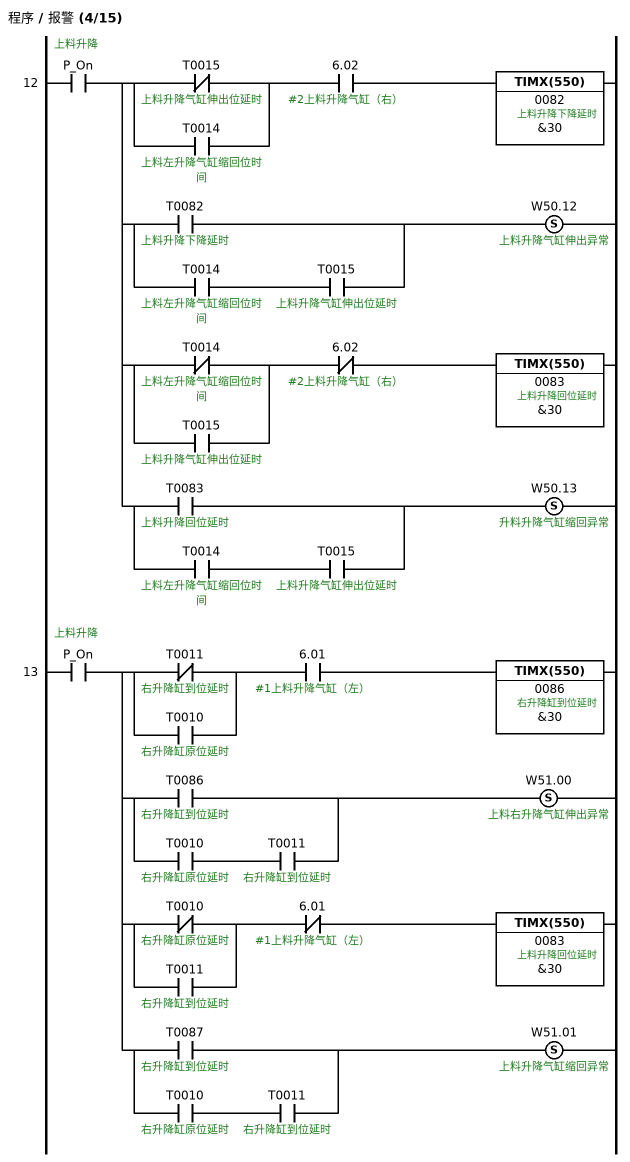
; rung 12: 上料升降
LD P_On
OUT TR0
LDNOT T0015  ; 上料升降气缸伸出位延时
OR T0014  ; 上料左升降气缸缩回位时间
ANDLD
AND 6.02  ; #2上料升降气缸（右）
TIMX(550) 0082 &30  ; 上料升降下降延时
LD TR0
LD T0082  ; 上料升降下降延时
LD T0014  ; 上料左升降气缸缩回位时间
AND T0015  ; 上料升降气缸伸出位延时
ORLD
ANDLD
SET W50.12  ; 上料升降气缸伸出异常
LD TR0
LDNOT T0014  ; 上料左升降气缸缩回位时间
OR T0015  ; 上料升降气缸伸出位延时
ANDLD
ANDNOT 6.02  ; #2上料升降气缸（右）
TIMX(550) 0083 &30  ; 上料升降回位延时
LD TR0
LD T0083  ; 上料升降回位延时
LD T0014  ; 上料左升降气缸缩回位时间
AND T0015  ; 上料升降气缸伸出位延时
ORLD
ANDLD
SET W50.13  ; 升料升降气缸缩回异常
; rung 13: 上料升降
LD P_On
OUT TR0
LDNOT T0011  ; 右升降缸到位延时
OR T0010  ; 右升降缸原位延时
ANDLD
AND 6.01  ; #1上料升降气缸（左）
TIMX(550) 0086 &30  ; 右升降缸到位延时
LD TR0
LD T0086  ; 右升降缸到位延时
LD T0010  ; 右升降缸原位延时
AND T0011  ; 右升降缸到位延时
ORLD
ANDLD
SET W51.00  ; 上料右升降气缸伸出异常
LD TR0
LDNOT T0010  ; 右升降缸原位延时
OR T0011  ; 右升降缸到位延时
ANDLD
ANDNOT 6.01  ; #1上料升降气缸（左）
TIMX(550) 0083 &30  ; 上料升降回位延时
LD TR0
LD T0087  ; 右升降缸到位延时
LD T0010  ; 右升降缸原位延时
AND T0011  ; 右升降缸到位延时
ORLD
ANDLD
SET W51.01  ; 上料升降气缸缩回异常

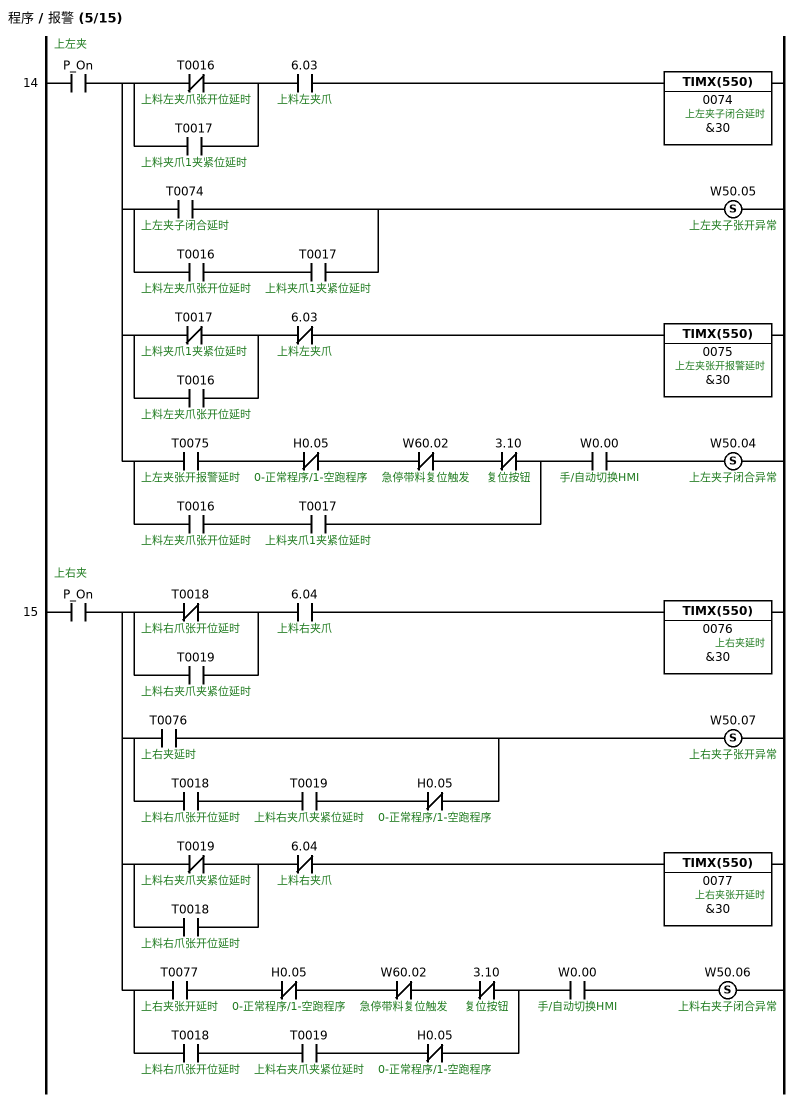
; rung 14: 上左夹
LD P_On
OUT TR0
LDNOT T0016  ; 上料左夹爪张开位延时
OR T0017  ; 上料夹爪1夹紧位延时
ANDLD
AND 6.03  ; 上料左夹爪
TIMX(550) 0074 &30  ; 上左夹子闭合延时
LD TR0
LD T0074  ; 上左夹子闭合延时
LD T0016  ; 上料左夹爪张开位延时
AND T0017  ; 上料夹爪1夹紧位延时
ORLD
ANDLD
SET W50.05  ; 上左夹子张开异常
LD TR0
LDNOT T0017  ; 上料夹爪1夹紧位延时
OR T0016  ; 上料左夹爪张开位延时
ANDLD
ANDNOT 6.03  ; 上料左夹爪
TIMX(550) 0075 &30  ; 上左夹张开报警延时
LD TR0
LD T0075  ; 上左夹张开报警延时
ANDNOT H0.05  ; 0-正常程序/1-空跑程序
ANDNOT W60.02  ; 急停带料复位触发
ANDNOT 3.10  ; 复位按钮
LD T0016  ; 上料左夹爪张开位延时
AND T0017  ; 上料夹爪1夹紧位延时
ORLD
ANDLD
AND W0.00  ; 手/自动切换HMI
SET W50.04  ; 上左夹子闭合异常
; rung 15: 上右夹
LD P_On
OUT TR0
LDNOT T0018  ; 上料右爪张开位延时
OR T0019  ; 上料右夹爪夹紧位延时
ANDLD
AND 6.04  ; 上料右夹爪
TIMX(550) 0076 &30  ; 上右夹延时
LD TR0
LD T0076  ; 上右夹延时
LD T0018  ; 上料右爪张开位延时
AND T0019  ; 上料右夹爪夹紧位延时
ANDNOT H0.05  ; 0-正常程序/1-空跑程序
ORLD
ANDLD
SET W50.07  ; 上右夹子张开异常
LD TR0
LDNOT T0019  ; 上料右夹爪夹紧位延时
OR T0018  ; 上料右爪张开位延时
ANDLD
ANDNOT 6.04  ; 上料右夹爪
TIMX(550) 0077 &30  ; 上右夹张开延时
LD TR0
LD T0077  ; 上右夹张开延时
ANDNOT H0.05  ; 0-正常程序/1-空跑程序
ANDNOT W60.02  ; 急停带料复位触发
ANDNOT 3.10  ; 复位按钮
LD T0018  ; 上料右爪张开位延时
AND T0019  ; 上料右夹爪夹紧位延时
ANDNOT H0.05  ; 0-正常程序/1-空跑程序
ORLD
ANDLD
AND W0.00  ; 手/自动切换HMI
SET W50.06  ; 上料右夹子闭合异常

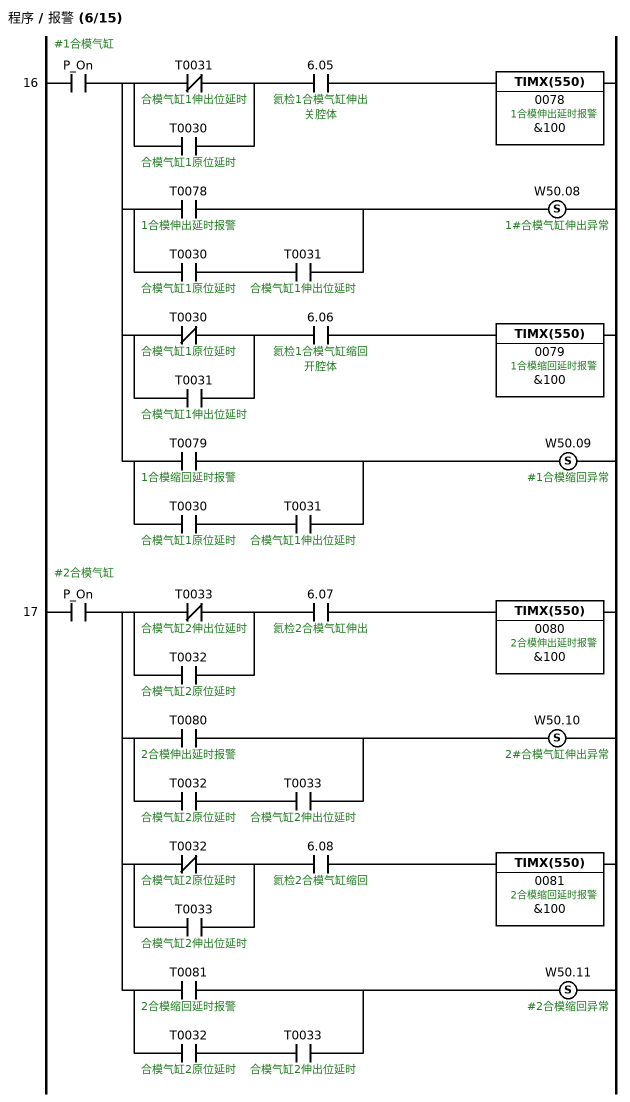
; rung 16: #1合模气缸
LD P_On
OUT TR0
LDNOT T0031  ; 合模气缸1伸出位延时
OR T0030  ; 合模气缸1原位延时
ANDLD
AND 6.05  ; 氦检1合模气缸伸出 关腔体
TIMX(550) 0078 &100  ; 1合模伸出延时报警
LD TR0
LD T0078  ; 1合模伸出延时报警
LD T0030  ; 合模气缸1原位延时
AND T0031  ; 合模气缸1伸出位延时
ORLD
ANDLD
SET W50.08  ; 1#合模气缸伸出异常
LD TR0
LDNOT T0030  ; 合模气缸1原位延时
OR T0031  ; 合模气缸1伸出位延时
ANDLD
AND 6.06  ; 氦检1合模气缸缩回 开腔体
TIMX(550) 0079 &100  ; 1合模缩回延时报警
LD TR0
LD T0079  ; 1合模缩回延时报警
LD T0030  ; 合模气缸1原位延时
AND T0031  ; 合模气缸1伸出位延时
ORLD
ANDLD
SET W50.09  ; #1合模缩回异常
; rung 17: #2合模气缸
LD P_On
OUT TR0
LDNOT T0033  ; 合模气缸2伸出位延时
OR T0032  ; 合模气缸2原位延时
ANDLD
AND 6.07  ; 氦检2合模气缸伸出
TIMX(550) 0080 &100  ; 2合模伸出延时报警
LD TR0
LD T0080  ; 2合模伸出延时报警
LD T0032  ; 合模气缸2原位延时
AND T0033  ; 合模气缸2伸出位延时
ORLD
ANDLD
SET W50.10  ; 2#合模气缸伸出异常
LD TR0
LDNOT T0032  ; 合模气缸2原位延时
OR T0033  ; 合模气缸2伸出位延时
ANDLD
AND 6.08  ; 氦检2合模气缸缩回
TIMX(550) 0081 &100  ; 2合模缩回延时报警
LD TR0
LD T0081  ; 2合模缩回延时报警
LD T0032  ; 合模气缸2原位延时
AND T0033  ; 合模气缸2伸出位延时
ORLD
ANDLD
SET W50.11  ; #2合模缩回异常

